(* IEC 61131-3 sources: programs/VI-54/VI-54_20171205/VI-54_20171205/Stations/Screen/LseClass170718/Class/EventUserInput, 1 file *)

(* ---- EventUserInput.st ---- *)
// Eigenschaften der Buffer
//----------------------------------------------------------------------------------------------------------------------------

#define   EventUser_MaxBufferLength     200           // Maximale Anzahl an Zeichen

(*!
<Class
	Name               = "EventUserInput"
	Revision           = "1.1"
	RealtimeTask       = "false"
	CyclicTask         = "false"
	BackgroundTask     = "false"
	Sigmatek           = "false"
	OSInterface        = "false"
	HighPriority       = "false"
	Automatic          = "false"
	UpdateMode         = "Prescan"
	SharedCommandTable = "true"
	Objectsize         = "(540,240)"
	Comment            = "class to create a user-input for the the EventJournal ">
	<Channels>
		<Server Name="OpenInput" Visualized="true" Initialize="false" WriteProtected="false" Retentive="false" Comment="write() will open the toucheditorwindow for input"/>
		<Client Name="coEventQueue" Required="true" Internal="false" Comment="object channel to EventQueue"/>
		<Client Name="coSystemLogging" Required="false" Internal="false" Comment="object channel to SystemLogging (optional)"/>
		<Client Name="StringEventUser" Required="true" Internal="true"/>
	</Channels>
	<RevDoku>
		<Owner Company="Sigmatek" Author="KaiAnd"/>
		<Dokumentation Revision="1.1" Date="2016-08-30" Author="KaiAnd" Company="Sigmatek" Description="changed procedure to get the name of the own object - the object name no longer must be &quot;EventUserInput1&quot;!"/>
		<Dokumentation Revision="1.0" Date="2016-05-20" Author="KaiAnd" Company="Sigmatek" Description="created; for user-input into the EventJournal"/>
	</RevDoku>
	<Network Name="EventUserInput">
		<!-- List of Components in this network -->
		<Components>
			<Object
				Name       = "_base"
				Class      = "_Global"
				Position   = "(120,120)"
				Visualized = "true"
				Remotely   = "true">
				<Channels>
					<Server Name="Server0"/>
					<Client Name="Lse"/>
				</Channels>
			</Object>
			<Object
				Name       = "StringEventUser"
				Class      = "String"
				Position   = "(120,360)"
				Visualized = "true"
				Remotely   = "true">
				<Channels>
					<Server Name="Data"/>
					<Client Name="SingleRealloc" Value="1"/>
				</Channels>
			</Object>
		</Components>
		<Comments>
		</Comments>
		<!-- List of Connections in this network -->
		<Connections>
			<Connection Source="this.Server0" Destination="_base.Server0" Vertices="(848,210),(420,210),"/>
			<Connection Source="_base.Lse" Destination="this.Lse" Vertices="(120,210),(38,210),"/>
			<Connection Source="this.StringEventUser" Destination="StringEventUser.Data"/>
		</Connections>
		<!-- Headerfiles -->
		<Options>
		</Options>
	</Network>
</Class>
*)
#pragma using _Global

EventUserInput : CLASS
: _Global
  //Servers:
	OpenInput 	: SvrCh_DINT;
  //Clients:
	StringEventUser 	: CltChCmd_String;
	coEventQueue 	: CltChCmd_EventQueue;
	coSystemLogging 	: CltChCmd_SystemLogging;
  //Variables:
		udVarNo_InpString 	: UDINT;
		IsCon_coSystemLogging 	: BOOL;
  //Functions:

	FUNCTION VIRTUAL GLOBAL Init;
				//! <Function Comment="methode will be called after lse-project is successfully loaded and &#13;&#10;possibly given communication to extern plc is stable" Name="IF_ProjectReady"/>
	FUNCTION VIRTUAL GLOBAL IF_ProjectReady
		VAR_INPUT
			state 	: BOOL;
		END_VAR
		VAR_OUTPUT
			retcode 	: BOOL;
		END_VAR;

	FUNCTION VIRTUAL GLOBAL IF_InputIsSaved
		VAR_INPUT
			pi 	: ^_INPUT;
			pr 	: ^_RESULT;
		END_VAR;

	FUNCTION VIRTUAL GLOBAL OpenInput::Write
		VAR_INPUT
			input (EAX) 	: DINT;
		END_VAR
		VAR_OUTPUT
			result (EAX) 	: DINT;
		END_VAR;
  //Tables:
	FUNCTION @STD
		VAR_OUTPUT
			ret_code	: CONFSTATES;
		END_VAR;
	FUNCTION GLOBAL TAB @CT_;
END_CLASS;

#pragma using String
#pragma usingLtd EventQueue
#pragma usingLtd SystemLogging

FUNCTION VIRTUAL GLOBAL EventUserInput::Init

  // Methode der Basis-Klasse
  _Global::Init();

  if (_FirstScan) then

    //---------------------------------------------------------------------------------------------
    //  check client-connnections and set flags
    //---------------------------------------------------------------------------------------------
    if (IsClientConnected(#coSystemLogging)) then
      IsCon_coSystemLogging := TRUE;
    else
      IsCon_coSystemLogging := FALSE;
    end_if;

  end_if;

END_FUNCTION

FUNCTION VIRTUAL GLOBAL EventUserInput::IF_ProjectReady
#pragma warning(disable:73); // disable warning
  VAR_INPUT
		state 	: BOOL;
  END_VAR
#pragma warning(default:73);
	VAR_OUTPUT
		retcode : BOOL;
	END_VAR
  VAR
    VarNoMe   : UDINT;
    dummy     : _UBYTE;
    myObjName : Array [0..99] of CHAR;   // ObjektName
  END_VAR

  //===============================================================================================
  //  Besorge eindeutige VAR-No des Strings für UserEvent-Input
  //===============================================================================================

  //---------------------------------------------------------------------------------------------
  //  den Namen des eigenen Objektes besorgen  V.1.1
  //---------------------------------------------------------------------------------------------
  VarNoMe := VarList_GetVarNoByID(x0:=this$udint, x1:=255, x2:=_FALSE);
  VarList_GetLabel(p0:=#myObjName[0], p1:=#dummy, x2:=VarNoMe);

  _strcat(dest:=#myObjName[0], src:="\StringEventUser.Data");   // Namen des eingebetteten String-Objektes anfügen

  //---------------------------------------------------------------------------------------------
  // VAR-No nun besorgen
  //---------------------------------------------------------------------------------------------
  udVarNo_InpString := VarList_GetVarNoStation(p0 := #myObjName[0], station := 255);

  retcode := TRUE;  // Retcode setzen, sonst kann Visu stehen bleiben

  //===============================================================================================

END_FUNCTION

FUNCTION VIRTUAL GLOBAL EventUserInput::OpenInput::Write
	VAR_INPUT
		input (EAX) 	: DINT;
	END_VAR
	VAR_OUTPUT
		result (EAX) 	: DINT;
	END_VAR

	OpenInput := input;
	result := OpenInput;

  //---------------------------------------------------------------------------------------
  //  Init Input
  //---------------------------------------------------------------------------------------
  StringEventUser.Clear();

  //---------------------------------------------------------------------------------------
  //  Command an LSE: öffne toucheditorwindow für Input auf angegebene VAR
  //---------------------------------------------------------------------------------------
  InsertCmd(x0 := CMD_EDITSERVER_HID,
            x1 := udVarNo_InpString$DINT,
            x2 := 0);

  //---------------------------------------------------------------------------------------

END_FUNCTION

FUNCTION VIRTUAL GLOBAL EventUserInput::IF_InputIsSaved
	VAR_INPUT
		pi 	: ^_INPUT;
		pr 	: ^_RESULT;
	END_VAR
  VAR
    tmpString       : ARRAY [0..EventUser_MaxBufferLength] OF _CHAR;
    tmpStringLength : UDINT;
  END_VAR

  //===============================================================================================
  //  auf "eigenen Input" reagieren (ASCII, eigene VAR-No)
  //===============================================================================================
  case pi^.io.typ of

    AS_ASCII:

      if ( (pi^.io.variable.info[0].state = VAR_VAL) &
           (pi^.io.variable.info[0].value = udVarNo_InpString$DINT) ) then

        tmpStringLength := StringEventUser.GetLength();
        if ((tmpStringLength > 0) & (tmpStringLength < EventUser_MaxBufferLength)) then

          //----- Event-String holen ----------------------------------------------------------
          StringEventUser.GetDataAt(pData:=#tmpString[0]$char, udSize:=tmpStringLength, udAt:=2);

          //----- Event-String eintragen ------------------------------------------------------
          if (coEventQueue.AddUserEvent(pEventString:=#tmpString[0]) = false) then

            if (IsCon_coSystemLogging = True) then
              coSystemLogging.LogEventText("EventQueue.AddUserEvent(): Benutzer-Event konnte nicht in EventJournal eingetragen werden");
            end_if;

          end_if;

        end_if;

      end_if;

  end_case;

  //===============================================================================================

END_FUNCTION
